INTERFACE ICylinder EXTENDS IBase

METHOD Extend : BOOL
VAR_INPUT
END_VAR
END_METHOD

METHOD Retract : BOOL
VAR_INPUT
END_VAR
END_METHOD

END_INTERFACE

(* stored: Version 1.1.0.1, ProductVersion 3.1.4024.12
   Itf ICylinder: Id {35407ab2-5bc7-4a54-b01b-ebe8fe750ff4}
   Method Extend: Id {434573bc-53df-45e3-90fd-53545f22a45e}
   Method Retract: Id {a89de3a3-2168-42aa-84d5-523c3d7d7268} *)
